(*

## Short summary

This interface provides assert statements for bit numbers:
For ``BYTE`` use `IBitNumberAssertions.short`
For ``WORD`` use `IBitNumberAssertions.simple`
For ``DWORD`` use `IBitNumberAssertions.double`
For ``LWORD`` use `IBitNumberAssertions.long`
For ``__XWORD`` use `IBitNumberAssertions.x`

.. <legal notes>

legal notes
=================
| SPDX-FileCopyrightText: © 2022 ekvip automation GmbH <info@ekvip.de>
| SPDX-License-Identifier: Apache-2.0
| For details check: Apache-2.0_

.. _Apache-2.0: https://www.apache.org/licenses/LICENSE-2.0

.. </legal notes>

properties
==================

*)

INTERFACE IBitNumberAssertions EXTENDS __SYSTEM.IQueryInterface

(*

## Short summary
Returns the interface `IDwordAssertions`
with assert statements for double words ``DWORD`` 

.. <legal notes>

legal notes
=================
| SPDX-FileCopyrightText: © 2022 ekvip automation GmbH <info@ekvip.de>
| SPDX-License-Identifier: Apache-2.0
| For details check: Apache-2.0_

.. _Apache-2.0: https://www.apache.org/licenses/LICENSE-2.0

.. </legal notes>

*)

PROPERTY double :IDwordAssertions
GET
END_GET
END_PROPERTY

(*

## Short summary
Returns the interface `ILwordAssertions`
with assert statements for long words ``LWORD`` 

.. <legal notes>

legal notes
=================
| SPDX-FileCopyrightText: © 2022 ekvip automation GmbH <info@ekvip.de>
| SPDX-License-Identifier: Apache-2.0
| For details check: Apache-2.0_

.. _Apache-2.0: https://www.apache.org/licenses/LICENSE-2.0

.. </legal notes>

*)

PROPERTY long :ILwordAssertions
GET
END_GET
END_PROPERTY

(*

## Short summary
Returns the interface `IByteAssertions`
with assert statements for bytes

.. <legal notes>

legal notes
=================
| SPDX-FileCopyrightText: © 2022 ekvip automation GmbH <info@ekvip.de>
| SPDX-License-Identifier: Apache-2.0
| For details check: Apache-2.0_

.. _Apache-2.0: https://www.apache.org/licenses/LICENSE-2.0

.. </legal notes>

*)

PROPERTY short :IByteAssertions
GET
END_GET
END_PROPERTY

(*

## Short summary
Returns the interface `IWordAssertions`
with assert statements for words 

.. <legal notes>

legal notes
=================
| SPDX-FileCopyrightText: © 2022 ekvip automation GmbH <info@ekvip.de>
| SPDX-License-Identifier: Apache-2.0
| For details check: Apache-2.0_

.. _Apache-2.0: https://www.apache.org/licenses/LICENSE-2.0

.. </legal notes>

*)

PROPERTY simple :IWordAssertions
GET
END_GET
END_PROPERTY

(*

## Short summary
Returns the interface `IXwordAssertions`
with assert statements for register length words ``__XWORD``

.. <legal notes>

legal notes
=================
| SPDX-FileCopyrightText: © 2022 ekvip automation GmbH <info@ekvip.de>
| SPDX-License-Identifier: Apache-2.0
| For details check: Apache-2.0_

.. _Apache-2.0: https://www.apache.org/licenses/LICENSE-2.0

.. </legal notes>

*)

PROPERTY x :IXwordAssertions
GET
END_GET
END_PROPERTY

END_INTERFACE

(* stored: Version 1.1.0.1, ProductVersion 3.1.4024.11
   Itf IBitNumberAssertions: Id {895eff78-c4a0-4ee1-bf26-cc1689b19a34}
   Property double: Id {be1b6755-03f0-4cbb-a198-494b2784a469}
   Get Get: Id {9bb9bd76-3cd4-45fa-bebb-9931a6ea8f2b}
   Property long: Id {587dc4f8-0531-41fd-91e8-27e69dd7baa7}
   Get Get: Id {3adf3dfa-6af4-46d9-bdf0-3cee1a719f38}
   Property short: Id {f4237945-ec7b-48b7-9410-edfa9257f61f}
   Get Get: Id {eb6215df-d0dd-4ad2-bd11-9c7cc998a599}
   Property simple: Id {3b50a78e-7cc9-4c5d-88fa-05ea12958332}
   Get Get: Id {a567337e-c9e4-4dbf-b73f-96f3c582ef2c}
   Property x: Id {94c1e8bf-9196-429a-ac21-956783054882}
   Get Get: Id {da951896-3f43-4dbd-8832-1e48c115dcc3} *)
